FUNCTION_BLOCK xPPU_PAC
VAR_INPUT
	i_error: POINTER TO ErrorManager;
	i_process: POINTER TO ProcessManager;
	i_state: POINTER TO StateTracker;
END_VAR
VAR
	m_emptyParams: ParameterSet;
	m_subRes: EOperationResult;
END_VAR

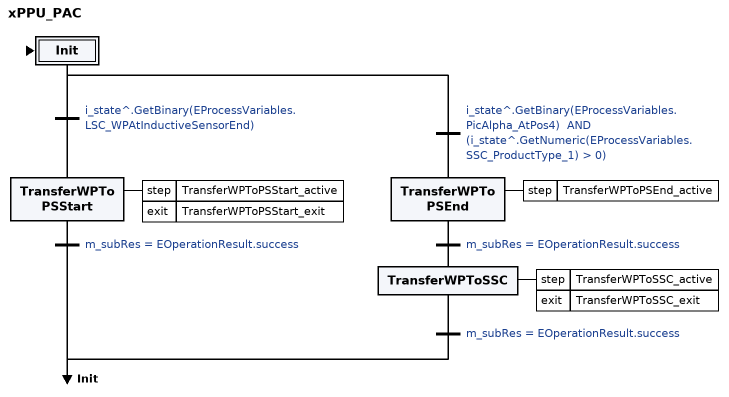
INITIAL_STEP Init:
END_STEP
TRANSITION FROM Init TO TransferWPToPSStart
    := i_state^.GetBinary(EProcessVariables.LSC_WPAtInductiveSensorEnd);
END_TRANSITION
STEP TransferWPToPSStart:
    TransferWPToPSStart_active(N);  // step action
    TransferWPToPSStart_exit(P0);  // exit action
END_STEP
TRANSITION FROM TransferWPToPSStart TO Init
    := m_subRes = EOperationResult.success;
END_TRANSITION
TRANSITION FROM Init TO TransferWPToPSEnd
    := i_state^.GetBinary(EProcessVariables.PicAlpha_AtPos4) AND (i_state^.GetNumeric(EProcessVariables.SSC_ProductType_1) > 0);
END_TRANSITION
STEP TransferWPToPSEnd:
    TransferWPToPSEnd_active(N);  // step action
END_STEP
TRANSITION FROM TransferWPToPSEnd TO TransferWPToSSC
    := m_subRes = EOperationResult.success;
END_TRANSITION
STEP TransferWPToSSC:
    TransferWPToSSC_active(N);  // step action
    TransferWPToSSC_exit(P0);  // exit action
END_STEP
TRANSITION FROM TransferWPToSSC TO Init
    := m_subRes = EOperationResult.success;
END_TRANSITION

ACTION TransferWPToPSEnd_active:
m_subRes := i_process^.Execute(
	EBehaviorType.control_primitive,
	EPrimitives.PAC_TransferWorkpieceTo_PSEnd,
	m_emptyParams);
END_ACTION

ACTION TransferWPToPSStart_active:
m_subRes := i_process^.Execute(
	EBehaviorType.control_primitive,
	EPrimitives.PAC_TransferWorkpieceTo_PSStart,
	m_emptyParams);
END_ACTION

ACTION TransferWPToPSStart_exit:
CASE LREAL_TO_INT(i_state^.GetNumeric(EProcessVariables.PAC_WPNumber)) OF
	1:	i_state^.ShiftProduct(EProducts.LSC_product, EProducts.PAC_product1);
	2:	i_state^.ShiftProduct(EProducts.LSC_product, EProducts.PAC_product2);
	3: 	i_state^.ShiftProduct(EProducts.LSC_product, EProducts.PAC_product3);
END_CASE
END_ACTION

ACTION TransferWPToSSC_active:
m_subRes := i_process^.Execute(
	EBehaviorType.control_primitive,
	EPrimitives.PAC_TransferWorkpieceTo_SSC,
	m_emptyParams);
END_ACTION

ACTION TransferWPToSSC_exit:
//shift products from PAC to SSC
i_state^.ShiftProduct(EProducts.PAC_product1, EProducts.SSC_product1);
i_state^.ShiftProduct(EProducts.PAC_product2, EProducts.SSC_product2);
END_ACTION

END_FUNCTION_BLOCK

(* stored: Version 1.1.0.1, ProductVersion 3.1.4024.4
   POU xPPU_PAC: Id {31492fc4-cd6a-47c9-9b47-d0d720b462dd}, SpecialFunc None
   Action TransferWPToPSEnd_active: Id {9967c60b-0391-4f00-8866-2458c7ebf309}
   Action TransferWPToPSStart_active: Id {d68f1288-0b40-43c1-94e0-2cb29ef010b6}
   Action TransferWPToPSStart_exit: Id {e95729a1-7980-4cdb-a261-cce4fad2646c}
   Action TransferWPToSSC_active: Id {b9f26b4d-03d2-4116-99c7-0e371a34fdf6}
   Action TransferWPToSSC_exit: Id {459563bc-8582-4e63-b8e6-b2dbdd8392c2} *)
